FUNCTION_BLOCK MaterialStorage
VAR_OUTPUT
	slots : ARRAY[1..GVL.maxQueue] OF STRING;
	//units : ARRAY[0..GVL.maxQueue] OF INT;
	
	empty AT %I* : ARRAY[1..GVL.maxQueue] OF BOOL;
END_VAR

METHOD findSlot : BOOL
VAR_INPUT
	materialID : STRING;
END_VAR
VAR_OUTPUT
	atSlot : INT := -1;
END_VAR
VAR
	i : INT;
END_VAR
IF materialID = '' THEN
	RETURN;
END_IF

FOR i:=0 TO GVL.maxQueue BY 1 DO
	IF slots[i] = materialID THEN
		atSlot := i;
		findSlot := TRUE;
		RETURN;
	END_IF
END_FOR
END_METHOD

METHOD getSlotsAsArray : POINTER TO STRING
getSlotsAsArray := ADR(slots);
END_METHOD

METHOD setupSlots : BOOL
VAR_INPUT
	setSlots : REFERENCE TO ARRAY[1..GVL.maxQueue] OF STRING;
END_VAR
slots := setSlots;
END_METHOD

END_FUNCTION_BLOCK

(* stored: Version 1.1.0.1, ProductVersion 3.1.4024.11
   POU MaterialStorage: Id {dcd61309-37ee-4727-afc9-669fba533248}, SpecialFunc None
   Method findSlot: Id {f0786625-8c57-43b6-af34-67307c7a7bb3}
   Method getSlotsAsArray: Id {80137db6-c2d9-4f11-ad61-62688f3299e7}
   Method setupSlots: Id {f8762705-6a29-4d8f-9219-4df3d8551e27} *)
